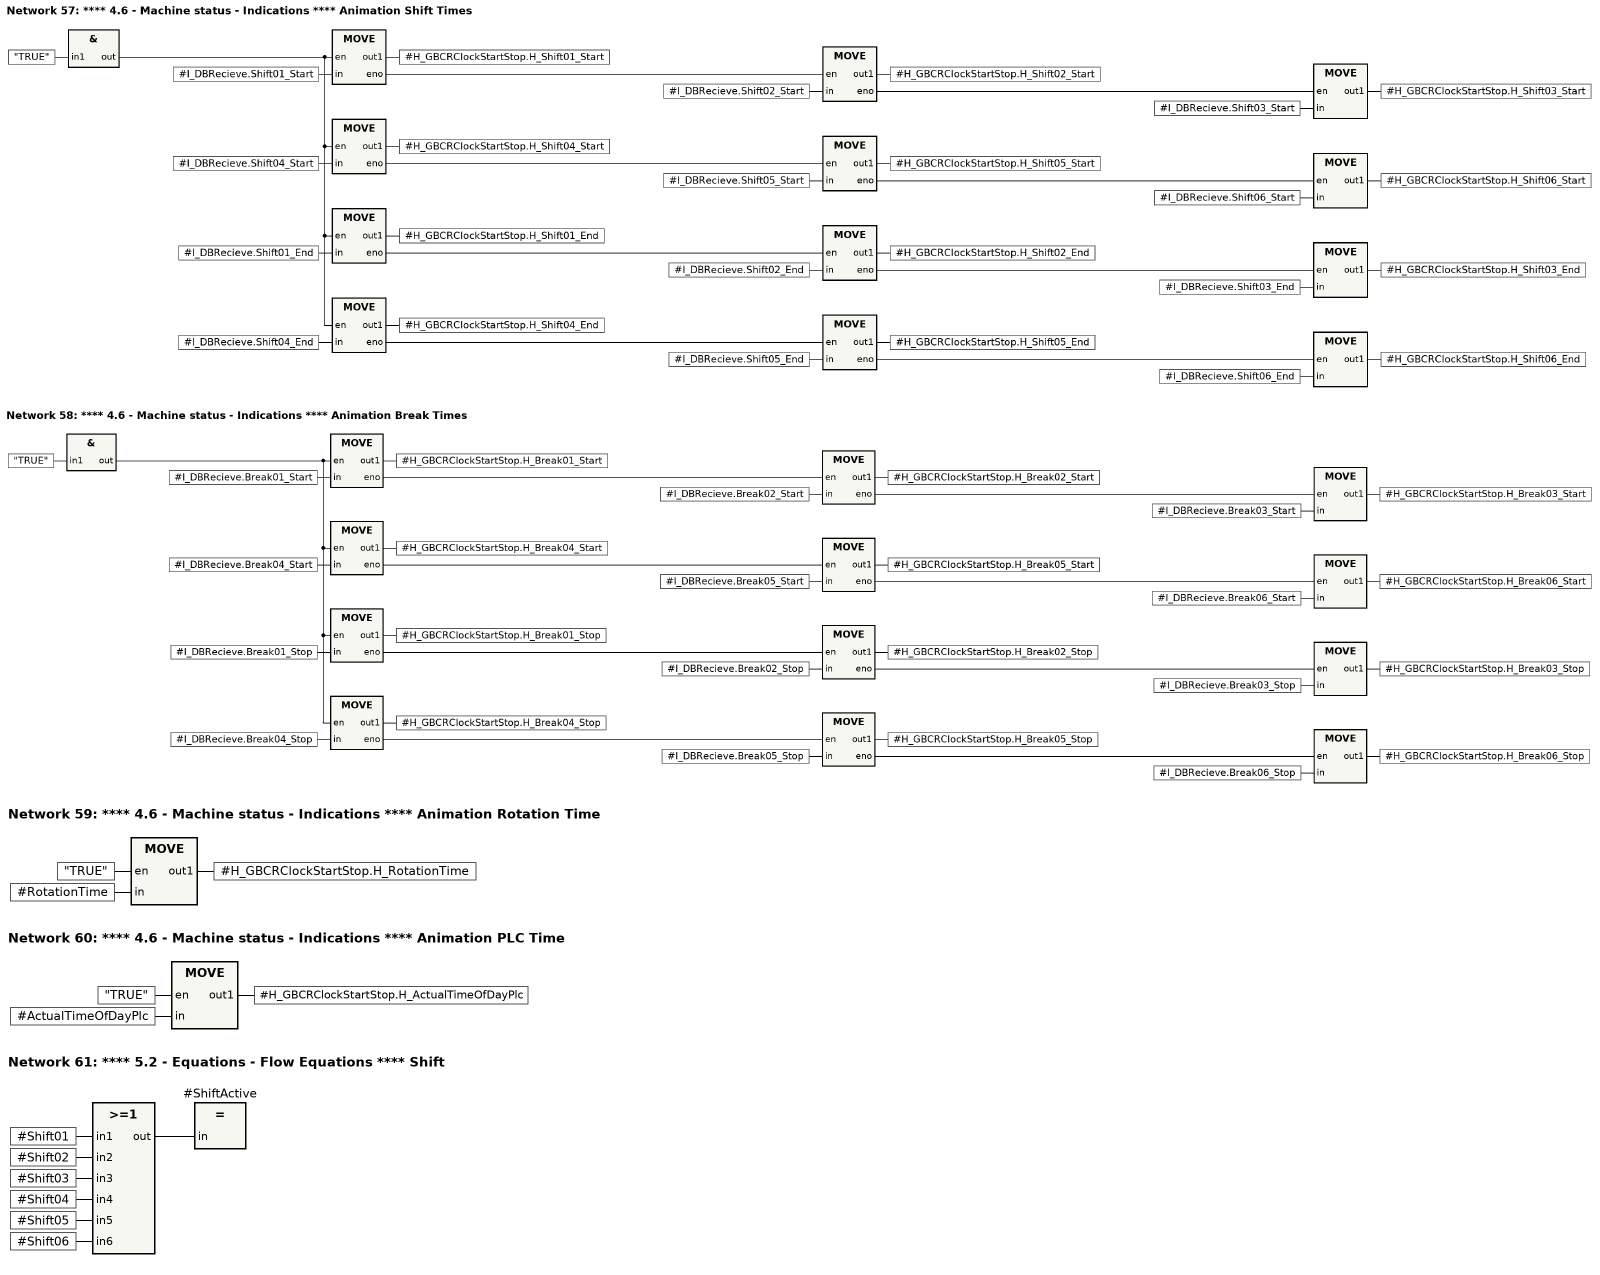
   IF "TRUE" THEN
       #H_GBCRClockStartStop.H_Shift01_Start := #I_DBRecieve.Shift01_Start;
       #H_GBCRClockStartStop.H_Shift02_Start := #I_DBRecieve.Shift02_Start;
       #H_GBCRClockStartStop.H_Shift03_Start := #I_DBRecieve.Shift03_Start;
       #H_GBCRClockStartStop.H_Shift04_Start := #I_DBRecieve.Shift04_Start;
       #H_GBCRClockStartStop.H_Shift05_Start := #I_DBRecieve.Shift05_Start;
       #H_GBCRClockStartStop.H_Shift06_Start := #I_DBRecieve.Shift06_Start;
       #H_GBCRClockStartStop.H_Shift01_End := #I_DBRecieve.Shift01_End;
       #H_GBCRClockStartStop.H_Shift02_End := #I_DBRecieve.Shift02_End;
       #H_GBCRClockStartStop.H_Shift03_End := #I_DBRecieve.Shift03_End;
       #H_GBCRClockStartStop.H_Shift04_End := #I_DBRecieve.Shift04_End;
       #H_GBCRClockStartStop.H_Shift05_End := #I_DBRecieve.Shift05_End;
       #H_GBCRClockStartStop.H_Shift06_End := #I_DBRecieve.Shift06_End;
   END_IF;
END_REGION

REGION Network 58: **** 4.6 - Machine status - Indications **** Animation Break Times
   IF "TRUE" THEN
       #H_GBCRClockStartStop.H_Break01_Start := #I_DBRecieve.Break01_Start;
       #H_GBCRClockStartStop.H_Break02_Start := #I_DBRecieve.Break02_Start;
       #H_GBCRClockStartStop.H_Break03_Start := #I_DBRecieve.Break03_Start;
       #H_GBCRClockStartStop.H_Break04_Start := #I_DBRecieve.Break04_Start;
       #H_GBCRClockStartStop.H_Break05_Start := #I_DBRecieve.Break05_Start;
       #H_GBCRClockStartStop.H_Break06_Start := #I_DBRecieve.Break06_Start;
       #H_GBCRClockStartStop.H_Break01_Stop := #I_DBRecieve.Break01_Stop;
       #H_GBCRClockStartStop.H_Break02_Stop := #I_DBRecieve.Break02_Stop;
       #H_GBCRClockStartStop.H_Break03_Stop := #I_DBRecieve.Break03_Stop;
       #H_GBCRClockStartStop.H_Break04_Stop := #I_DBRecieve.Break04_Stop;
       #H_GBCRClockStartStop.H_Break05_Stop := #I_DBRecieve.Break05_Stop;
       #H_GBCRClockStartStop.H_Break06_Stop := #I_DBRecieve.Break06_Stop;
   END_IF;
END_REGION

REGION Network 59: **** 4.6 - Machine status - Indications **** Animation Rotation Time
   IF "TRUE" THEN #H_GBCRClockStartStop.H_RotationTime := #RotationTime; END_IF;
END_REGION

REGION Network 60: **** 4.6 - Machine status - Indications **** Animation PLC Time
   IF "TRUE" THEN #H_GBCRClockStartStop.H_ActualTimeOfDayPlc := #ActualTimeOfDayPlc; END_IF;
END_REGION

REGION Network 61: **** 5.2 - Equations - Flow Equations **** Shift
   #ShiftActive := #Shift01 OR #Shift02 OR #Shift03 OR #Shift04 OR #Shift05 OR #Shift06;
END_REGION

REGION Network 62: **** 5.2 - Equations - Flow Equations **** Break
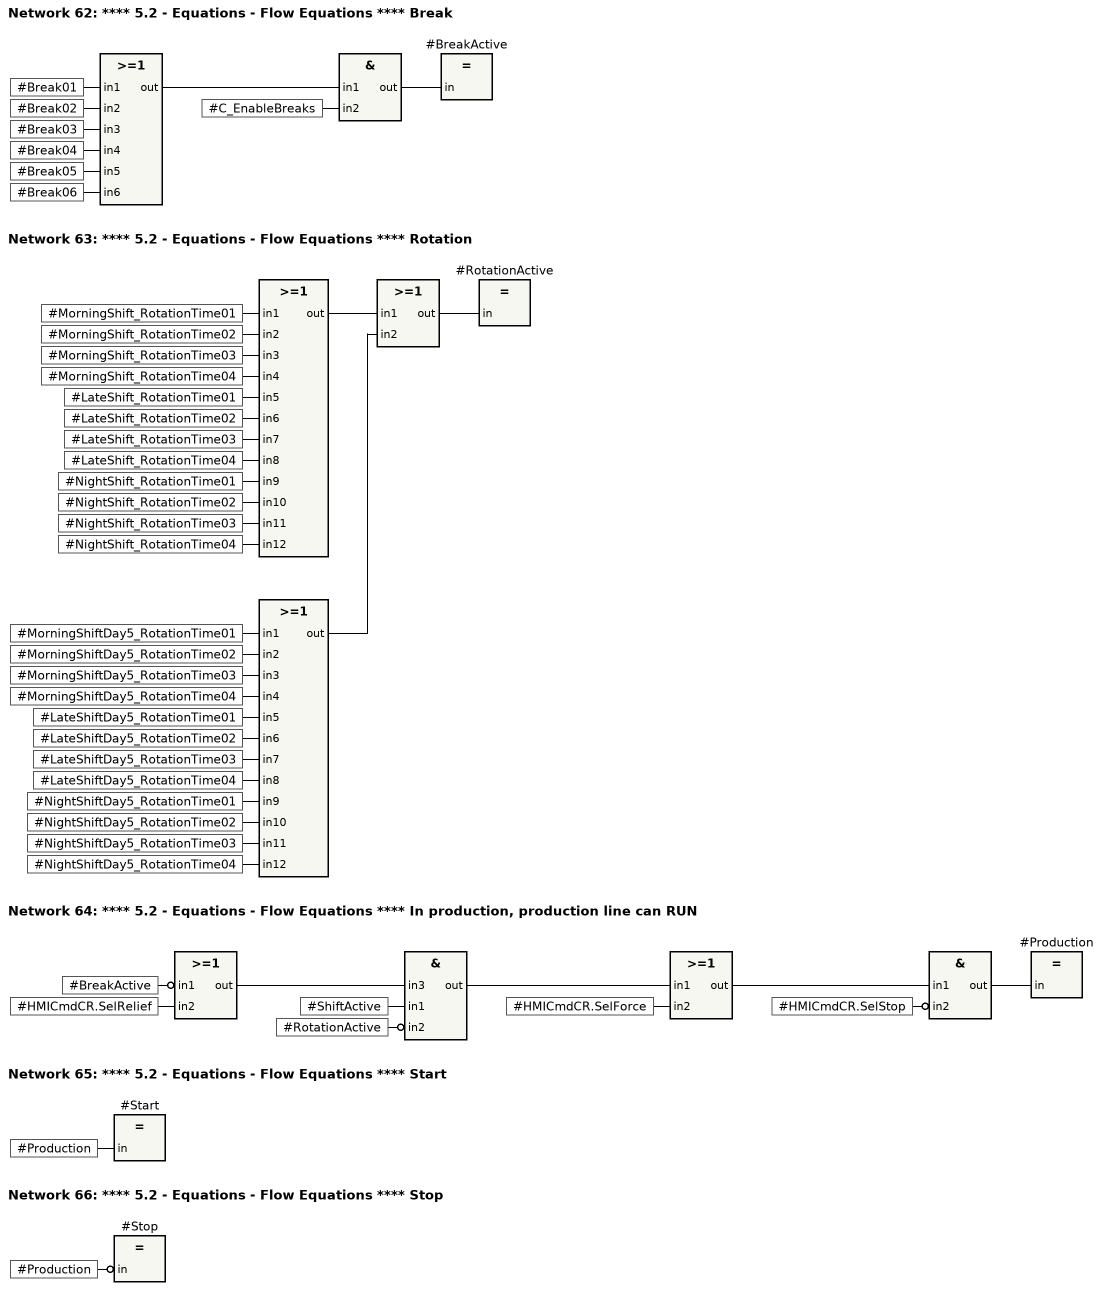
   #BreakActive := (#Break01 OR #Break02 OR #Break03 OR #Break04 OR #Break05 OR #Break06) AND #C_EnableBreaks;
END_REGION

REGION Network 63: **** 5.2 - Equations - Flow Equations **** Rotation
   #RotationActive := #MorningShift_RotationTime01 OR #MorningShift_RotationTime02 OR #MorningShift_RotationTime03 OR #MorningShift_RotationTime04 OR #LateShift_RotationTime01 OR #LateShift_RotationTime02 OR #LateShift_RotationTime03 OR #LateShift_RotationTime04 OR #NightShift_RotationTime01 OR #NightShift_RotationTime02 OR #NightShift_RotationTime03 OR #NightShift_RotationTime04 OR #MorningShiftDay5_RotationTime01 OR #MorningShiftDay5_RotationTime02 OR #MorningShiftDay5_RotationTime03 OR #MorningShiftDay5_RotationTime04 OR #LateShiftDay5_RotationTime01 OR #LateShiftDay5_RotationTime02 OR #LateShiftDay5_RotationTime03 OR #LateShiftDay5_RotationTime04 OR #NightShiftDay5_RotationTime01 OR #NightShiftDay5_RotationTime02 OR #NightShiftDay5_RotationTime03 OR #NightShiftDay5_RotationTime04;
END_REGION

REGION Network 64: **** 5.2 - Equations - Flow Equations **** In production, production line can RUN
   #Production := (((NOT #BreakActive OR #HMICmdCR.SelRelief) AND #ShiftActive AND NOT #RotationActive) OR #HMICmdCR.SelForce) AND NOT #HMICmdCR.SelStop;
END_REGION

REGION Network 65: **** 5.2 - Equations - Flow Equations **** Start
   #Start := #Production;
END_REGION

REGION Network 66: **** 5.2 - Equations - Flow Equations **** Stop
   #Stop := NOT #Production;
END_REGION

REGION Network 67: **** 8 - Outputs **** Start production line
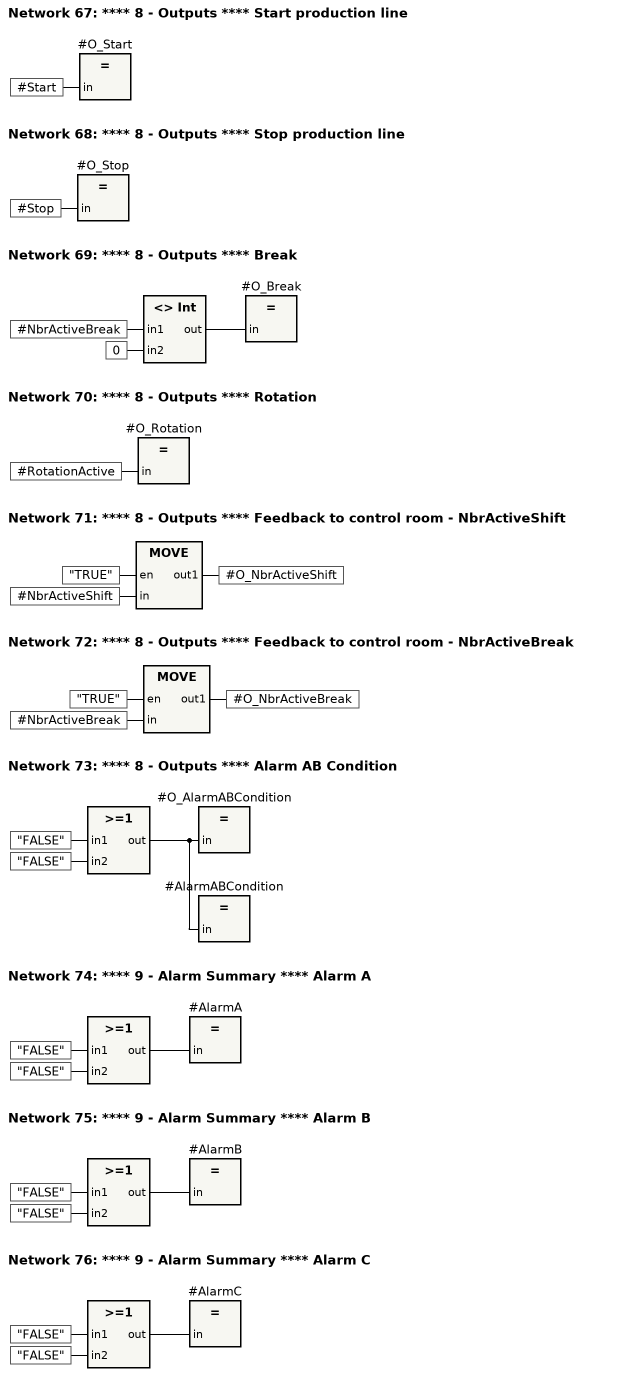
   #O_Start := #Start;
END_REGION

REGION Network 68: **** 8 - Outputs **** Stop production line
   #O_Stop := #Stop;
END_REGION

REGION Network 69: **** 8 - Outputs **** Break
   #O_Break := #NbrActiveBreak <> 0;
END_REGION

REGION Network 70: **** 8 - Outputs **** Rotation
   #O_Rotation := #RotationActive;
END_REGION

REGION Network 71: **** 8 - Outputs **** Feedback to control room - NbrActiveShift
   IF "TRUE" THEN #O_NbrActiveShift := #NbrActiveShift; END_IF;
END_REGION

REGION Network 72: **** 8 - Outputs **** Feedback to control room - NbrActiveBreak
   IF "TRUE" THEN #O_NbrActiveBreak := #NbrActiveBreak; END_IF;
END_REGION

REGION Network 73: **** 8 - Outputs **** Alarm AB Condition
   // Alarm AB Condition
   #O_AlarmABCondition := "FALSE" OR "FALSE";
   #AlarmABCondition := #O_AlarmABCondition;
END_REGION

REGION Network 74: **** 9 - Alarm Summary **** Alarm A
   // Alarm A
   #AlarmA := "FALSE" OR "FALSE";
END_REGION

REGION Network 75: **** 9 - Alarm Summary **** Alarm B
   // Alarm B
   #AlarmB := "FALSE" OR "FALSE";
END_REGION

REGION Network 76: **** 9 - Alarm Summary **** Alarm C
   // Alarm C
   #AlarmC := "FALSE" OR "FALSE";
END_REGION

REGION Network 77: **** 9 - Alarm Summary **** Alarm D
   // Alarm D
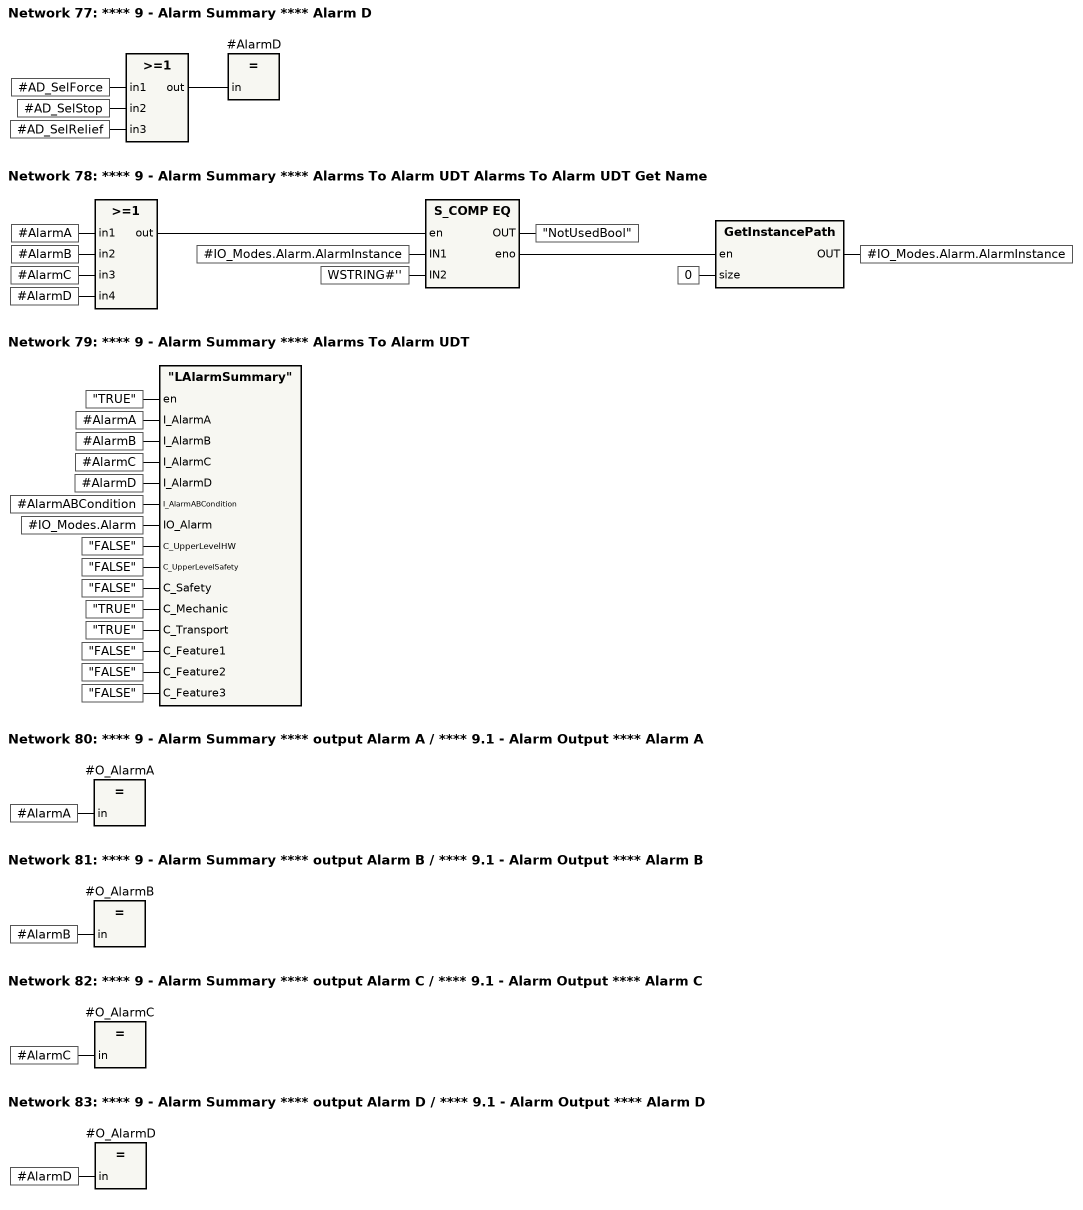
   #AlarmD := #AD_SelForce OR #AD_SelStop OR #AD_SelRelief;
END_REGION

REGION Network 78: **** 9 - Alarm Summary **** Alarms To Alarm UDT Alarms To Alarm UDT Get Name
   // Alarm / Alarm D
   S_COMP(EN := #AlarmA OR #AlarmB OR #AlarmC OR #AlarmD,
          IN1 := #IO_Modes.Alarm.AlarmInstance,
          IN2 := WSTRING#'',
          OUT => "NotUsedBool",
          ENO => #_w1);
   IF #_w1 THEN GetInstancePath(size := 0, OUT => #IO_Modes.Alarm.AlarmInstance); END_IF;
END_REGION

REGION Network 79: **** 9 - Alarm Summary **** Alarms To Alarm UDT
   // Alarm / Alarm D
   IF "TRUE" THEN
       "LAlarmSummary"(I_AlarmA := #AlarmA,
                       I_AlarmB := #AlarmB,
                       I_AlarmC := #AlarmC,
                       I_AlarmD := #AlarmD,
                       I_AlarmABCondition := #AlarmABCondition,
                       IO_Alarm := #IO_Modes.Alarm,
                       C_UpperLevelHW := "FALSE",
                       C_UpperLevelSafety := "FALSE",
                       C_Safety := "FALSE",
                       C_Mechanic := "TRUE",
                       C_Transport := "TRUE",
                       C_Feature1 := "FALSE",
                       C_Feature2 := "FALSE",
                       C_Feature3 := "FALSE");
   END_IF;
END_REGION

REGION Network 80: **** 9 - Alarm Summary **** output Alarm A / **** 9.1 - Alarm Output **** Alarm A
   // Alarm A
   #O_AlarmA := #AlarmA;
END_REGION

REGION Network 81: **** 9 - Alarm Summary **** output Alarm B / **** 9.1 - Alarm Output **** Alarm B
   // Alarm B
   #O_AlarmB := #AlarmB;
END_REGION

REGION Network 82: **** 9 - Alarm Summary **** output Alarm C / **** 9.1 - Alarm Output **** Alarm C
   // Alarm C
   #O_AlarmC := #AlarmC;
END_REGION

REGION Network 83: **** 9 - Alarm Summary **** output Alarm D / **** 9.1 - Alarm Output **** Alarm D
   // Alarm D
   #O_AlarmD := #AlarmD;
END_REGION

REGION Network 84: **** 9 - Alarm Summary **** output Alarm Word / **** 9.2 - Alarm DWord**** Alarm To DWord
   // Alarm To Word
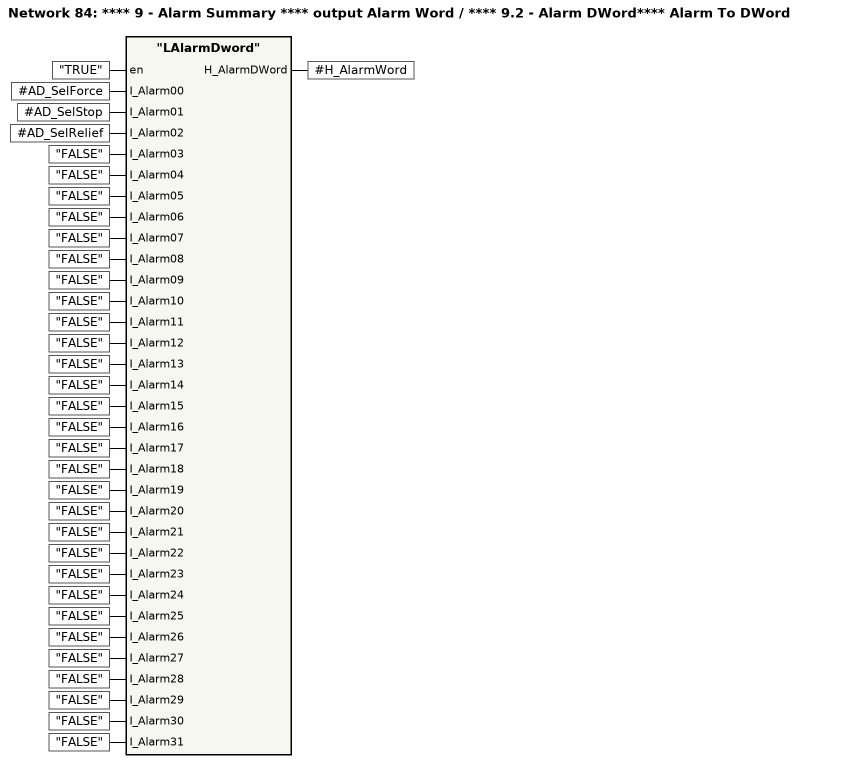
   IF "TRUE" THEN
       "LAlarmDword"(I_Alarm00 := #AD_SelForce,
                     I_Alarm01 := #AD_SelStop,
                     I_Alarm02 := #AD_SelRelief,
                     I_Alarm03 := "FALSE",
                     I_Alarm04 := "FALSE",
                     I_Alarm05 := "FALSE",
                     I_Alarm06 := "FALSE",
                     I_Alarm07 := "FALSE",
                     I_Alarm08 := "FALSE",
                     I_Alarm09 := "FALSE",
                     I_Alarm10 := "FALSE",
                     I_Alarm11 := "FALSE",
                     I_Alarm12 := "FALSE",
                     I_Alarm13 := "FALSE",
                     I_Alarm14 := "FALSE",
                     I_Alarm15 := "FALSE",
                     I_Alarm16 := "FALSE",
                     I_Alarm17 := "FALSE",
                     I_Alarm18 := "FALSE",
                     I_Alarm19 := "FALSE",
                     I_Alarm20 := "FALSE",
                     I_Alarm21 := "FALSE",
                     I_Alarm22 := "FALSE",
                     I_Alarm23 := "FALSE",
                     I_Alarm24 := "FALSE",
                     I_Alarm25 := "FALSE",
                     I_Alarm26 := "FALSE",
                     I_Alarm27 := "FALSE",
                     I_Alarm28 := "FALSE",
                     I_Alarm29 := "FALSE",
                     I_Alarm30 := "FALSE",
                     I_Alarm31 := "FALSE",
                     H_AlarmDWord => #H_AlarmWord);
   END_IF;
END_REGION
END_FUNCTION_BLOCK
